// TIA Portal project "TcpTest01(two_close_loop_ok)" (V15)

(* hardware
DEVICE "S7-1200 station_1"  S7-1200 Station
   slot 0: "Rack_0"  S7-1200 Rack  Rack  V1.0
   slot 1: "PLC_1"  CPU 1214C DC/DC/Rly  6ES7 214-1HG40-0XB0  V4.0
   slot 2: "AQ 4x14BIT_1"  6ES7 232-4HD32-0XB0  V2.0
   slot 3: "AI 4x13BIT_1"  6ES7 231-4HD32-0XB0  V2.0
   slot 101: "CM 1241 (RS422/485)_1"  6ES7 241-1CH32-0XB0  V2.2
*)

// ===== PLC "PLC_1"  CPU 1214C DC/DC/Rly =====

VAR_GLOBAL   // PLC tag table "默认变量表"
   "System_Byte" AT %MB1 : Byte;
   "FirstScan" AT %M1.0 : Bool;
   "DiagStatusUpdate" AT %M1.1 : Bool;
   "AlwaysTRUE" AT %M1.2 : Bool;
   "AlwaysFALSE" AT %M1.3 : Bool;
   "Clock_Byte" AT %MB0 : Byte;
   "Clock_10Hz" AT %M0.0 : Bool;
   "Clock_5Hz" AT %M0.1 : Bool;
   "Clock_2.5Hz" AT %M0.2 : Bool;
   "Clock_2Hz" AT %M0.3 : Bool;
   "Clock_1.25Hz" AT %M0.4 : Bool;
   "Clock_1Hz" AT %M0.5 : Bool;
   "Clock_0.625Hz" AT %M0.6 : Bool;
   "Clock_0.5Hz" AT %M0.7 : Bool;
   "AD0" AT %IW64 : Int;
   "AD1" AT %IW66 : Int;
   "DA0" AT %QW96 : Int;
   "DA1" AT %QW98 : Int;
   "DA2" AT %QW100 : Int;
   "AD1_1" AT %IW112 : Int;
   "AD1_2" AT %IW114 : Int;
   "AD1_3" AT %IW116 : Int;
   "AD1_4" AT %IW118 : Int;
END_VAR

DATA_BLOCK "REAL_TO_BYTE_DB"   // DB1
{ S7_Optimized_Access := 'TRUE' }
VERSION : 0.1
// stored: InstanceOfName REAL_TO_BYTE
"REAL_TO_BYTE"
BEGIN
END_DATA_BLOCK

DATA_BLOCK "REAL_TO_BYTE_DB_2#"   // DB2
{ S7_Optimized_Access := 'TRUE' }
VERSION : 0.1
// stored: InstanceOfName REAL_TO_BYTE
"REAL_TO_BYTE"
BEGIN
END_DATA_BLOCK

DATA_BLOCK "BYTE_TO_REAL_DB"   // DB3
{ S7_Optimized_Access := 'TRUE' }
VERSION : 0.1
// stored: InstanceOfName BYTE_TO_REAL
"BYTE_TO_REAL"
BEGIN
END_DATA_BLOCK

DATA_BLOCK "TcpDB_1"   // DB4
{ S7_Optimized_Access := 'TRUE' }
VERSION : 0.1
   VAR
      SendBuf0 : Array[0..11] of Byte;
   END_VAR
BEGIN
END_DATA_BLOCK

DATA_BLOCK "BYTE_TO_REAL_DB_1"   // DB5
{ S7_Optimized_Access := 'TRUE' }
VERSION : 0.1
// stored: InstanceOfName BYTE_TO_REAL
"BYTE_TO_REAL"
BEGIN
END_DATA_BLOCK

DATA_BLOCK "BYTE_TO_REAL_DB_2"   // DB14
{ S7_Optimized_Access := 'TRUE' }
VERSION : 0.1
// stored: InstanceOfName BYTE_TO_REAL
"BYTE_TO_REAL"
BEGIN
END_DATA_BLOCK

DATA_BLOCK "REAL_TO_BYTE_DB_1"   // DB29
{ S7_Optimized_Access := 'TRUE' }
VERSION : 0.1
// stored: InstanceOfName REAL_TO_BYTE
"REAL_TO_BYTE"
BEGIN
END_DATA_BLOCK

DATA_BLOCK "REAL_TO_BYTE_DB_1#"   // DB30
{ S7_Optimized_Access := 'TRUE' }
VERSION : 0.1
// stored: InstanceOfName REAL_TO_BYTE
"REAL_TO_BYTE"
BEGIN
END_DATA_BLOCK

DATA_BLOCK "REAL_TO_BYTE_DB_3#"   // DB31
{ S7_Optimized_Access := 'TRUE' }
VERSION : 0.1
// stored: InstanceOfName REAL_TO_BYTE
"REAL_TO_BYTE"
BEGIN
END_DATA_BLOCK

DATA_BLOCK "REAL_TO_BYTE_DB_2"   // DB32
{ S7_Optimized_Access := 'TRUE' }
VERSION : 0.1
// stored: InstanceOfName REAL_TO_BYTE
"REAL_TO_BYTE"
BEGIN
END_DATA_BLOCK

DATA_BLOCK "BYTE_TO_DWORD_DB"   // DB38
{ S7_Optimized_Access := 'TRUE' }
VERSION : 0.1
// stored: InstanceOfName BYTE_TO_DWORD
"BYTE_TO_DWORD"
BEGIN
END_DATA_BLOCK

FUNCTION_BLOCK "BYTE_TO_REAL"   // FB1, LAD
{ S7_Optimized_Access := 'TRUE' }
VERSION : 0.1
   VAR_INPUT
      i : Int;
      receiveBufIn : Array[0..11] of Byte;
   END_VAR
   VAR_OUTPUT
      convRealOut : Real;
   END_VAR
   VAR_TEMP
      convDwordTemp0 : DWord;
      convDwordTemp1 : DWord;
      convDwordTemp2 : DWord;
      convDwordTemp3 : DWord;
      convDwordTemp4 : DWord;
      k0 : Int;
      k1 : Int;
      k2 : Int;
      k3 : Int;
   END_VAR
BEGIN

REGION Network 1
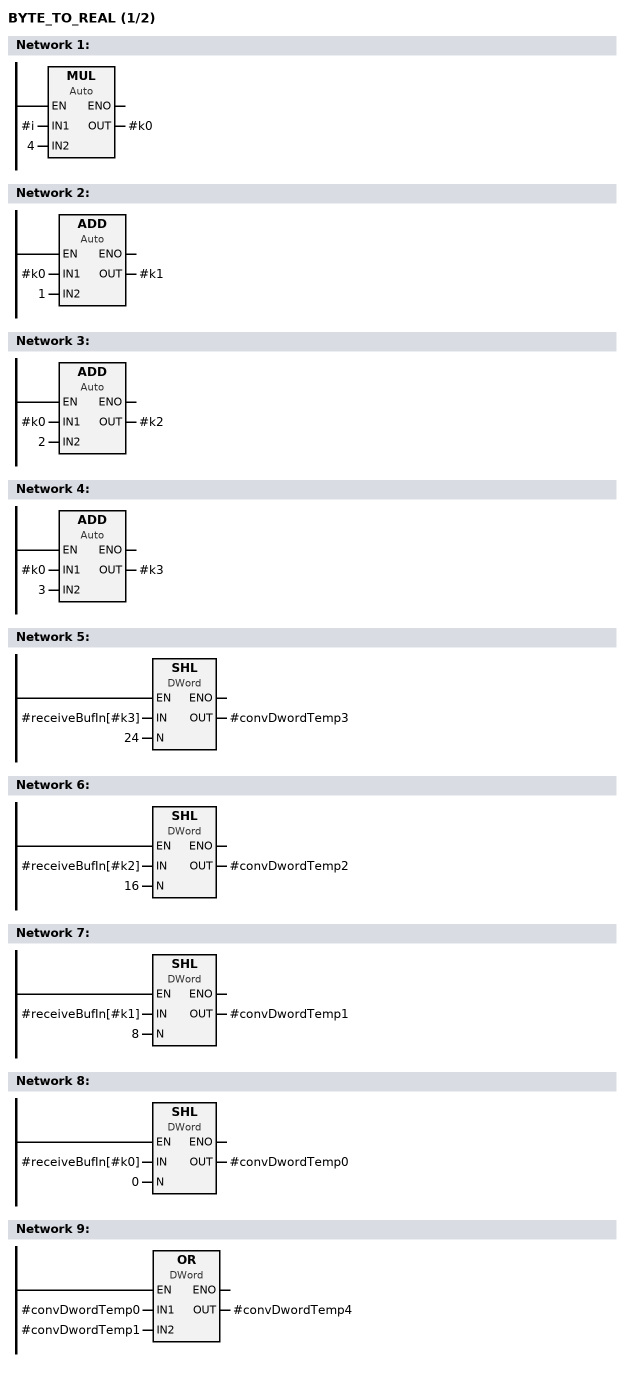
   RUNG wire#powerrail
      Mul(in1 := #i, in2 := 4, out => #k0)
   END_RUNG
   // the same network as SCL:
   #k0 := #i * 4;
END_REGION

REGION Network 2
   RUNG wire#powerrail
      Add(in1 := #k0, in2 := 1, out => #k1)
   END_RUNG
   // the same network as SCL:
   #k1 := #k0 + 1;
END_REGION

REGION Network 3
   RUNG wire#powerrail
      Add(in1 := #k0, in2 := 2, out => #k2)
   END_RUNG
   // the same network as SCL:
   #k2 := #k0 + 2;
END_REGION

REGION Network 4
   RUNG wire#powerrail
      Add(in1 := #k0, in2 := 3, out => #k3)
   END_RUNG
   // the same network as SCL:
   #k3 := #k0 + 3;
END_REGION

REGION Network 5
   RUNG wire#powerrail
      { S7_Templates := "SrcType := DWord" } Shl(in := #receiveBufIn[#k3], n := 24, out => #convDwordTemp3)
   END_RUNG
   // the same network as SCL:
   #convDwordTemp3 := SHL(IN := #receiveBufIn[#k3], N := 24);
END_REGION

REGION Network 6
   RUNG wire#powerrail
      { S7_Templates := "SrcType := DWord" } Shl(in := #receiveBufIn[#k2], n := 16, out => #convDwordTemp2)
   END_RUNG
   // the same network as SCL:
   #convDwordTemp2 := SHL(IN := #receiveBufIn[#k2], N := 16);
END_REGION

REGION Network 7
   RUNG wire#powerrail
      { S7_Templates := "SrcType := DWord" } Shl(in := #receiveBufIn[#k1], n := 8, out => #convDwordTemp1)
   END_RUNG
   // the same network as SCL:
   #convDwordTemp1 := SHL(IN := #receiveBufIn[#k1], N := 8);
END_REGION

REGION Network 8
   RUNG wire#powerrail
      { S7_Templates := "SrcType := DWord" } Shl(in := #receiveBufIn[#k0], n := 0, out => #convDwordTemp0)
   END_RUNG
   // the same network as SCL:
   #convDwordTemp0 := SHL(IN := #receiveBufIn[#k0], N := 0);
END_REGION

REGION Network 9
   #convDwordTemp4 := #convDwordTemp0 OR #convDwordTemp1;
END_REGION

REGION Network 10
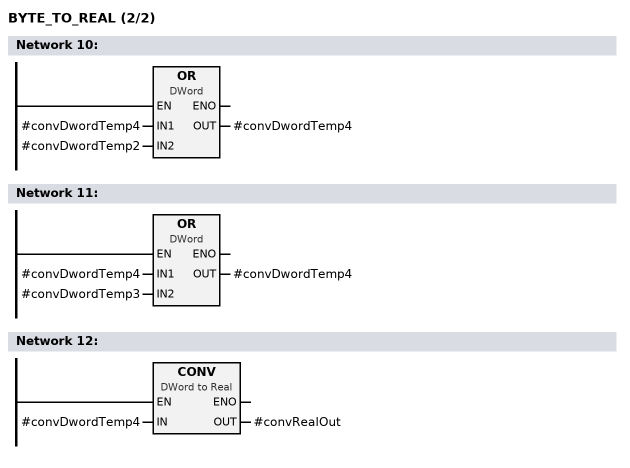
   #convDwordTemp4 := #convDwordTemp4 OR #convDwordTemp2;
END_REGION

REGION Network 11
   #convDwordTemp4 := #convDwordTemp4 OR #convDwordTemp3;
END_REGION

REGION Network 12
   RUNG wire#powerrail
      { S7_Templates := "[SrcType := DWord, DestType := Real]" } Convert(in := #convDwordTemp4, out => #convRealOut)
   END_RUNG
   // the same network as SCL:
   #convRealOut := DWORD_TO_REAL(#convDwordTemp4);
END_REGION
END_FUNCTION_BLOCK

FUNCTION_BLOCK "REAL_TO_BYTE"   // FB6, LAD
{ S7_Optimized_Access := 'TRUE' }
VERSION : 0.1
   VAR_INPUT
      i : Int;
      InputReal : Real;
   END_VAR
   VAR_TEMP
      OutputByte0 : Byte;
      OutputByte1 : Byte;
      OutputByte2 : Byte;
      OutputByte3 : Byte;
      convDwordTemp : DWord;
      convByteTemp0 : Byte;
      convByteTemp1 : Byte;
      convByteTemp2 : Byte;
      convByteTemp3 : Byte;
      k0 : Int;
      k1 : Int;
      k2 : Int;
      k3 : Int;
   END_VAR
BEGIN

REGION Network 1
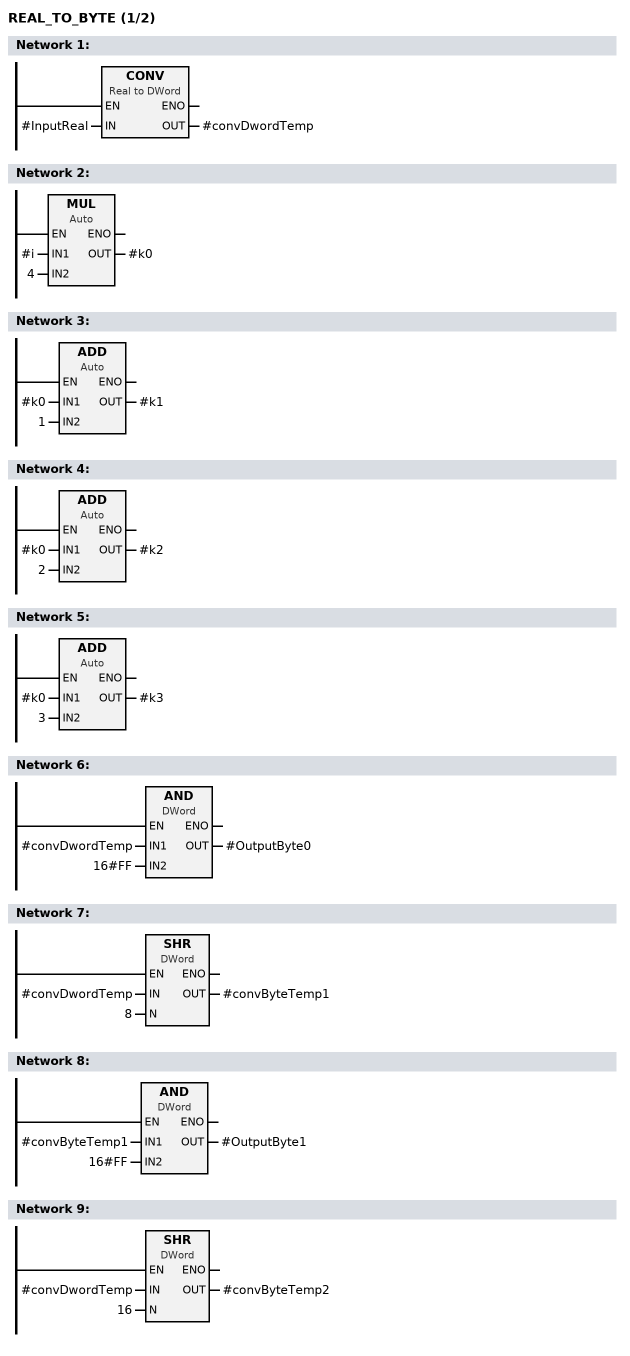
   RUNG wire#powerrail
      { S7_Templates := "[SrcType := Real, DestType := DWord]" } Convert(in := #InputReal, out => #convDwordTemp)
   END_RUNG
   // the same network as SCL:
   #convDwordTemp := REAL_TO_DWORD(#InputReal);
END_REGION

REGION Network 2
   RUNG wire#powerrail
      Mul(in1 := #i, in2 := 4, out => #k0)
   END_RUNG
   // the same network as SCL:
   #k0 := #i * 4;
END_REGION

REGION Network 3
   RUNG wire#powerrail
      Add(in1 := #k0, in2 := 1, out => #k1)
   END_RUNG
   // the same network as SCL:
   #k1 := #k0 + 1;
END_REGION

REGION Network 4
   RUNG wire#powerrail
      Add(in1 := #k0, in2 := 2, out => #k2)
   END_RUNG
   // the same network as SCL:
   #k2 := #k0 + 2;
END_REGION

REGION Network 5
   RUNG wire#powerrail
      Add(in1 := #k0, in2 := 3, out => #k3)
   END_RUNG
   // the same network as SCL:
   #k3 := #k0 + 3;
END_REGION

REGION Network 6
   RUNG wire#powerrail
      { S7_Templates := "SrcType := DWord" } And(in1 := #convDwordTemp, in2 := 16#FF, out => #OutputByte0)
   END_RUNG
   // the same network as SCL:
   #OutputByte0 := #convDwordTemp AND 16#FF;
END_REGION

REGION Network 7
   RUNG wire#powerrail
      { S7_Templates := "SrcType := DWord" } Shr(in := #convDwordTemp, n := 8, out => #convByteTemp1)
   END_RUNG
   // the same network as SCL:
   #convByteTemp1 := SHR(IN := #convDwordTemp, N := 8);
END_REGION

REGION Network 8
   RUNG wire#powerrail
      { S7_Templates := "SrcType := DWord" } And(in1 := #convByteTemp1, in2 := 16#FF, out => #OutputByte1)
   END_RUNG
   // the same network as SCL:
   #OutputByte1 := #convByteTemp1 AND 16#FF;
END_REGION

REGION Network 9
   RUNG wire#powerrail
      { S7_Templates := "SrcType := DWord" } Shr(in := #convDwordTemp, n := 16, out => #convByteTemp2)
   END_RUNG
   // the same network as SCL:
   #convByteTemp2 := SHR(IN := #convDwordTemp, N := 16);
END_REGION

REGION Network 10
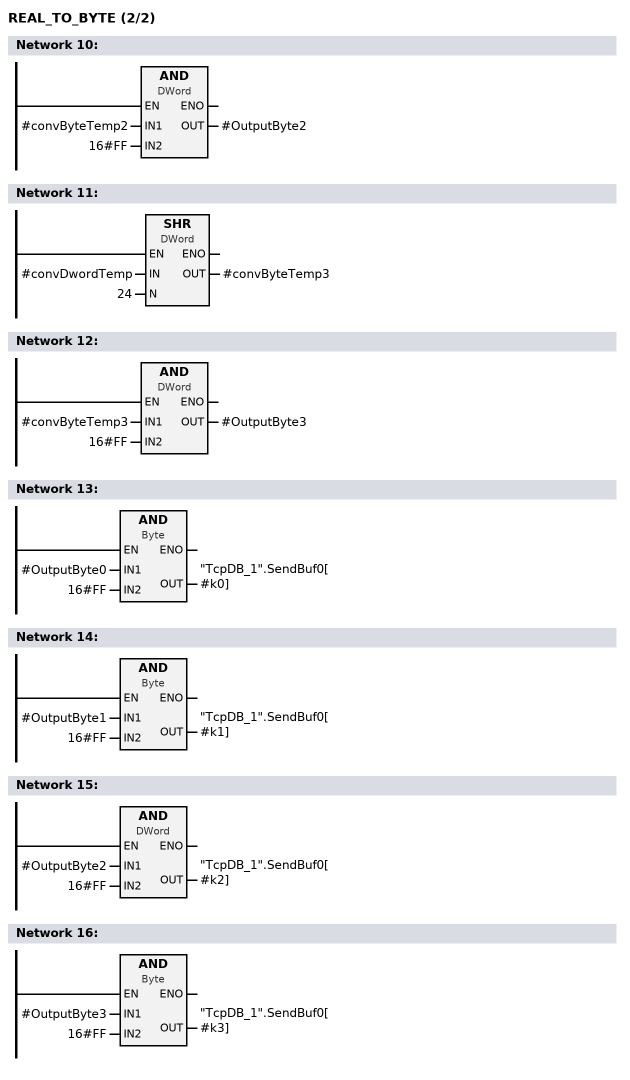
   RUNG wire#powerrail
      { S7_Templates := "SrcType := DWord" } And(in1 := #convByteTemp2, in2 := 16#FF, out => #OutputByte2)
   END_RUNG
   // the same network as SCL:
   #OutputByte2 := #convByteTemp2 AND 16#FF;
END_REGION

REGION Network 11
   RUNG wire#powerrail
      { S7_Templates := "SrcType := DWord" } Shr(in := #convDwordTemp, n := 24, out => #convByteTemp3)
   END_RUNG
   // the same network as SCL:
   #convByteTemp3 := SHR(IN := #convDwordTemp, N := 24);
END_REGION

REGION Network 12
   RUNG wire#powerrail
      { S7_Templates := "SrcType := DWord" } And(in1 := #convByteTemp3, in2 := 16#FF, out => #OutputByte3)
   END_RUNG
   // the same network as SCL:
   #OutputByte3 := #convByteTemp3 AND 16#FF;
END_REGION

REGION Network 13
   RUNG wire#powerrail
      { S7_Templates := "SrcType := Byte" } And(in1 := #OutputByte0, in2 := 16#FF, out => "TcpDB_1".SendBuf0[#k0])
   END_RUNG
   // the same network as SCL:
   "TcpDB_1".SendBuf0[#k0] := #OutputByte0 AND 16#FF;
END_REGION

REGION Network 14
   RUNG wire#powerrail
      { S7_Templates := "SrcType := Byte" } And(in1 := #OutputByte1, in2 := 16#FF, out => "TcpDB_1".SendBuf0[#k1])
   END_RUNG
   // the same network as SCL:
   "TcpDB_1".SendBuf0[#k1] := #OutputByte1 AND 16#FF;
END_REGION

REGION Network 15
   RUNG wire#powerrail
      { S7_Templates := "SrcType := DWord" } And(in1 := #OutputByte2, in2 := 16#FF, out => "TcpDB_1".SendBuf0[#k2])
   END_RUNG
   // the same network as SCL:
   "TcpDB_1".SendBuf0[#k2] := #OutputByte2 AND 16#FF;
END_REGION

REGION Network 16
   RUNG wire#powerrail
      { S7_Templates := "SrcType := Byte" } And(in1 := #OutputByte3, in2 := 16#FF, out => "TcpDB_1".SendBuf0[#k3])
   END_RUNG
   // the same network as SCL:
   "TcpDB_1".SendBuf0[#k3] := #OutputByte3 AND 16#FF;
END_REGION
END_FUNCTION_BLOCK

FUNCTION_BLOCK "BYTE_TO_DWORD"   // FB9, LAD
{ S7_Optimized_Access := 'TRUE' }
VERSION : 0.1
   VAR_INPUT
      i : Int;
      receiveBufIn : Array[0..1215] of Byte;
   END_VAR
   VAR_OUTPUT
      convDwordOut : DWord;
   END_VAR
   VAR_TEMP
      convDwordTemp0 : DWord;
      convDwordTemp1 : DWord;
      convDwordTemp2 : DWord;
      convDwordTemp3 : DWord;
      convDwordTemp4 : DWord;
      k0 : Int;
      k1 : Int;
      k2 : Int;
      k3 : Int;
   END_VAR
BEGIN

REGION Network 1
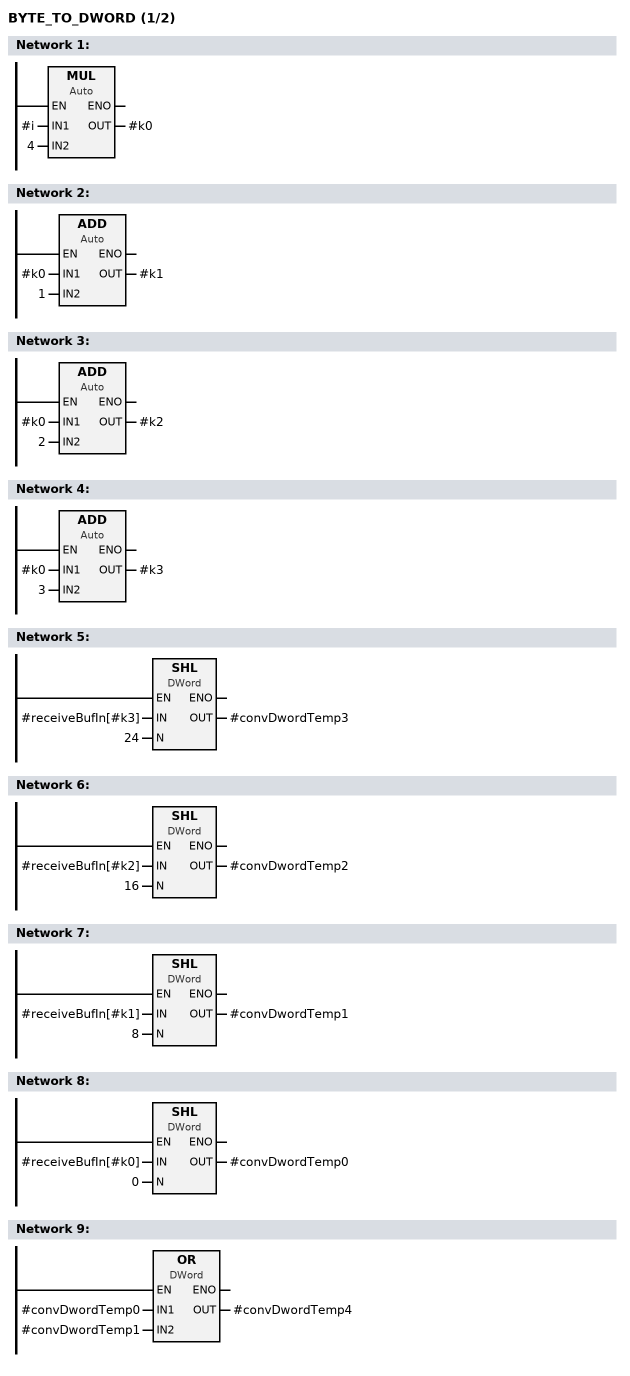
   RUNG wire#powerrail
      Mul(in1 := #i, in2 := 4, out => #k0)
   END_RUNG
   // the same network as SCL:
   #k0 := #i * 4;
END_REGION

REGION Network 2
   RUNG wire#powerrail
      Add(in1 := #k0, in2 := 1, out => #k1)
   END_RUNG
   // the same network as SCL:
   #k1 := #k0 + 1;
END_REGION

REGION Network 3
   RUNG wire#powerrail
      Add(in1 := #k0, in2 := 2, out => #k2)
   END_RUNG
   // the same network as SCL:
   #k2 := #k0 + 2;
END_REGION

REGION Network 4
   RUNG wire#powerrail
      Add(in1 := #k0, in2 := 3, out => #k3)
   END_RUNG
   // the same network as SCL:
   #k3 := #k0 + 3;
END_REGION

REGION Network 5
   RUNG wire#powerrail
      { S7_Templates := "SrcType := DWord" } Shl(in := #receiveBufIn[#k3], n := 24, out => #convDwordTemp3)
   END_RUNG
   // the same network as SCL:
   #convDwordTemp3 := SHL(IN := #receiveBufIn[#k3], N := 24);
END_REGION

REGION Network 6
   RUNG wire#powerrail
      { S7_Templates := "SrcType := DWord" } Shl(in := #receiveBufIn[#k2], n := 16, out => #convDwordTemp2)
   END_RUNG
   // the same network as SCL:
   #convDwordTemp2 := SHL(IN := #receiveBufIn[#k2], N := 16);
END_REGION

REGION Network 7
   RUNG wire#powerrail
      { S7_Templates := "SrcType := DWord" } Shl(in := #receiveBufIn[#k1], n := 8, out => #convDwordTemp1)
   END_RUNG
   // the same network as SCL:
   #convDwordTemp1 := SHL(IN := #receiveBufIn[#k1], N := 8);
END_REGION

REGION Network 8
   RUNG wire#powerrail
      { S7_Templates := "SrcType := DWord" } Shl(in := #receiveBufIn[#k0], n := 0, out => #convDwordTemp0)
   END_RUNG
   // the same network as SCL:
   #convDwordTemp0 := SHL(IN := #receiveBufIn[#k0], N := 0);
END_REGION

REGION Network 9
   #convDwordTemp4 := #convDwordTemp0 OR #convDwordTemp1;
END_REGION

REGION Network 10
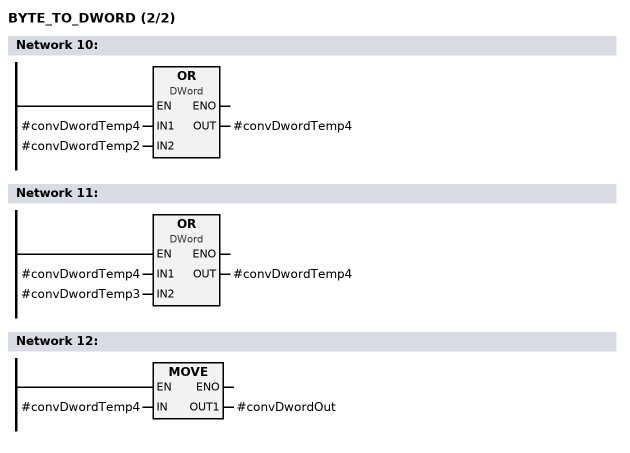
   #convDwordTemp4 := #convDwordTemp4 OR #convDwordTemp2;
END_REGION

REGION Network 11
   #convDwordTemp4 := #convDwordTemp4 OR #convDwordTemp3;
END_REGION

REGION Network 12
   RUNG wire#powerrail
      Move(in := #convDwordTemp4, out1 => #convDwordOut)
   END_RUNG
   // the same network as SCL:
   #convDwordOut := #convDwordTemp4;
END_REGION
END_FUNCTION_BLOCK

FUNCTION "BYTE_TO_DWORD_FC" : Void   // FC10, LAD
{ S7_Optimized_Access := 'TRUE' }
VERSION : 0.1
   VAR_INPUT
      i : Int;
      receiveBufIn : Array[0..1215] of Byte;
   END_VAR
   VAR_OUTPUT
      convDwordOut : DWord;
   END_VAR
   VAR_TEMP
      convDwordTemp0 : DWord;
      convDwordTemp1 : DWord;
      convDwordTemp2 : DWord;
      convDwordTemp3 : DWord;
      convDwordTemp4 : DWord;
      k0 : Int;
      k1 : Int;
      k2 : Int;
      k3 : Int;
   END_VAR
BEGIN

REGION Network 1
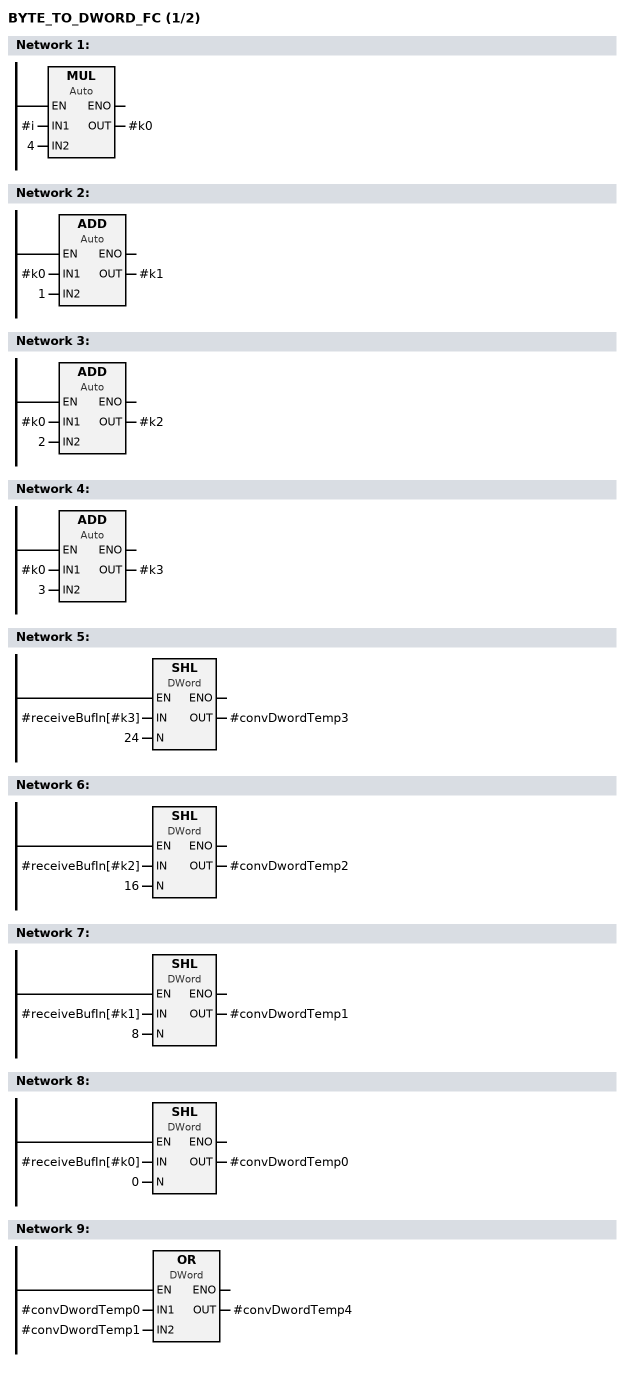
   RUNG wire#powerrail
      Mul(in1 := #i, in2 := 4, out => #k0)
   END_RUNG
   // the same network as SCL:
   #k0 := #i * 4;
END_REGION

REGION Network 2
   RUNG wire#powerrail
      Add(in1 := #k0, in2 := 1, out => #k1)
   END_RUNG
   // the same network as SCL:
   #k1 := #k0 + 1;
END_REGION

REGION Network 3
   RUNG wire#powerrail
      Add(in1 := #k0, in2 := 2, out => #k2)
   END_RUNG
   // the same network as SCL:
   #k2 := #k0 + 2;
END_REGION

REGION Network 4
   RUNG wire#powerrail
      Add(in1 := #k0, in2 := 3, out => #k3)
   END_RUNG
   // the same network as SCL:
   #k3 := #k0 + 3;
END_REGION

REGION Network 5
   RUNG wire#powerrail
      { S7_Templates := "SrcType := DWord" } Shl(in := #receiveBufIn[#k3], n := 24, out => #convDwordTemp3)
   END_RUNG
   // the same network as SCL:
   #convDwordTemp3 := SHL(IN := #receiveBufIn[#k3], N := 24);
END_REGION

REGION Network 6
   RUNG wire#powerrail
      { S7_Templates := "SrcType := DWord" } Shl(in := #receiveBufIn[#k2], n := 16, out => #convDwordTemp2)
   END_RUNG
   // the same network as SCL:
   #convDwordTemp2 := SHL(IN := #receiveBufIn[#k2], N := 16);
END_REGION

REGION Network 7
   RUNG wire#powerrail
      { S7_Templates := "SrcType := DWord" } Shl(in := #receiveBufIn[#k1], n := 8, out => #convDwordTemp1)
   END_RUNG
   // the same network as SCL:
   #convDwordTemp1 := SHL(IN := #receiveBufIn[#k1], N := 8);
END_REGION

REGION Network 8
   RUNG wire#powerrail
      { S7_Templates := "SrcType := DWord" } Shl(in := #receiveBufIn[#k0], n := 0, out => #convDwordTemp0)
   END_RUNG
   // the same network as SCL:
   #convDwordTemp0 := SHL(IN := #receiveBufIn[#k0], N := 0);
END_REGION

REGION Network 9
   #convDwordTemp4 := #convDwordTemp0 OR #convDwordTemp1;
END_REGION

REGION Network 10
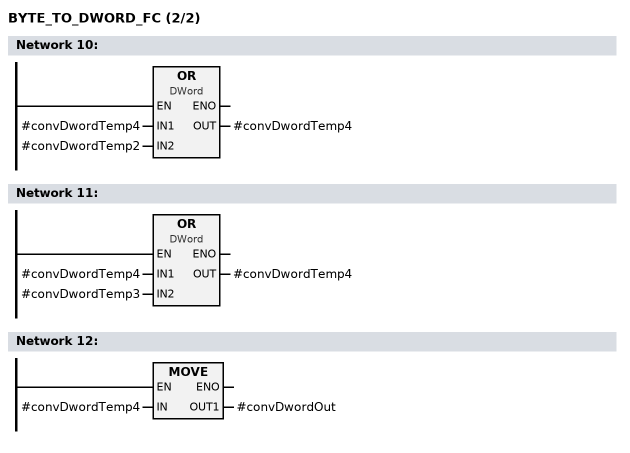
   #convDwordTemp4 := #convDwordTemp4 OR #convDwordTemp2;
END_REGION

REGION Network 11
   #convDwordTemp4 := #convDwordTemp4 OR #convDwordTemp3;
END_REGION

REGION Network 12
   RUNG wire#powerrail
      Move(in := #convDwordTemp4, out1 => #convDwordOut)
   END_RUNG
   // the same network as SCL:
   #convDwordOut := #convDwordTemp4;
END_REGION
END_FUNCTION